FUNCTION LoadFromMemory : BOOL
VAR_INPUT
    sData : REFERENCE TO STRING(2000);
END_VAR
VAR
    fbJson     : FB_JsonSaxReader;
    pJsonParse : FB_ReadJSON;
    //pJsonParse : FB_ReadRecipeJson;

    i : int;
END_VAR

// pJsonParse.myArrayInput1 REF= PERS.iStationTimeDef1;
// pJsonParse.myArrayInput2 REF= PERS.iStationTimeDef2;
fbJson.Parse(sJson := sData, ipHdl := pJsonParse);

END_FUNCTION

(* stored: Version 1.1.0.1, ProductVersion 3.1.4024.6
   POU LoadFromMemory: Id {34b1f23f-155f-4282-b68e-def4f76673a0}, SpecialFunc None *)
